FUNCTION_BLOCK fbChiniseMachine_v2_Laser IMPLEMENTS I_StationMachine
VAR_INPUT
	stSlaveParms				: stModTcpSlaveParams;
	bNextMachineWork			: BOOL;
	fbTCP_Send: REFERENCE TO FB_TCP_SendString;
	
END_VAR
VAR_OUTPUT
END_VAR
VAR
	I_PimSystem					: I_PIM;
	I_ModbusTcpCommunication 	: I_ModbusTcpCore;
	iWorkStep 					: INT;
	bServiceReset				: BOOL;
	stPimCommunicationData		: stPimMachineData;
	stModbusTcpData				: stModTcpQue;
	fbResetWaitTime				: TON;
	fbWorkEnded					: R_TRIG;					// Rising edgre reaction for end of cycle 
	iLastPartsRecord			: WORD;
	arReadArray					: ARRAY[0..GVL_ModbusTCP_Constants.iWriteRegisterLimit] OF INT;
	arWriteArray				: ARRAY[0..GVL_ModbusTCP_Constants.iWriteRegisterLimit] OF INT;
	rCommIntervalCounter		: REAL;
	nLastOperationStatus		: nModbusTCP_CommandStatus;
	fbCommunicationTimeout		: TON;
	bLastLifeBitState			: BOOL;
	stHMI						: stChiniseMachineHmiData;
	fbLifeBitPLC				: TON;
	stEthernetCommunication		: stInOutsEthernetCommunication;
	//Laser TCP
	fbLaserControl				:FB_LaserControl;
END_VAR

ACT_Background();
fbLaserControl(fbTCP_Send:=fbTCP_Send);

CASE iWorkStep OF
	0:	// Init
		iWorkStep := 5;
		
	5:	// Wait for next state
		I_PimSystem.mSetNewMachineState(nPIM_MachineStates._2_ReadyForNewOperation);	
		fbLaserControl.mRequestJobRefresh();
		iWorkStep := 10;
		
	10: // Start of work
		IF stPimCommunicationData.wGoodPartsAmount > iLastPartsRecord THEN
			IF I_PimSystem.mSetNewMachineState(nPIM_MachineStates._3_NewOperationStarted) THEN
				iLastPartsRecord := iLastPartsRecord +1;
				iWorkStep := 15;
				I_PimSystem.mSetNewMachineState(nPIM_MachineStates._4_OperationInProgress);
			END_IF
		END_IF
		IF fbLaserControl.stHMI_Laser.bEnableLaserTCPCOmmunication AND fbLaserControl.bJobRefreshError THEN
			mNewEvent(nEventClass:=nPIM_EventClasses.Error,nEvent:=nLaser_ErrorCodes.LaserTCPCommunicationError);
		END_IF
		
	15:	// Work ended
		iWorkStep := 5;
		I_PimSystem.mSetNewMachineState(nPIM_MachineStates._5_OperationEndedOK);
		
	90:	// Wysterowanie w przypadku błędu
		I_PimSystem.mSetNewMachineState(nPIM_MachineStates._8_WaitForReset);
		iWorkStep := 91;
		
	91:	// Oczekiwanie na reset
		IF I_PimSystem.mSetNewMachineState(nPIM_MachineStates._9_ResetInProgress) OR bServiceReset THEN
			bServiceReset := FALSE;
			stPimCommunicationData.bResetError := TRUE;
			fbCommunicationTimeout(IN:=FALSE);
			fbResetWaitTime(IN:=FALSE);
			iWorkStep := 92;
		END_IF
		
	92: // Wait some time
		fbResetWaitTime(IN:=TRUE,PT:=T#2S);
		IF fbResetWaitTime.Q THEN
			fbResetWaitTime(IN:=FALSE,PT:=T#2S);
			stPimCommunicationData.bResetError := FALSE;
			stPimCommunicationData.bConfirmError := TRUE;
			iWorkStep := 93;
		END_IF
		
	93:	// Check error state
		fbResetWaitTime(IN:=TRUE,PT:=T#2S);
		IF NOT stPimCommunicationData.bError THEN
			stPimCommunicationData.bConfirmError := FALSE;
			iWorkStep := 95;
			fbResetWaitTime(IN:=TRUE,PT:=T#2S);
		ELSIF fbResetWaitTime.Q THEN
			fbResetWaitTime(IN:=TRUE,PT:=T#2S);
			stPimCommunicationData.bResetError := FALSE;
			stPimCommunicationData.bConfirmError := FALSE;
			mNewEvent(nEventClass:=nPIM_EventClasses.Error,nEvent:=stPimCommunicationData.iErrorCode+stSlaveParms.iErrorOffset);
		END_IF
		
	95: // Potwierdzenie błędu itp
		I_PimSystem.mSetNewMachineState(nPIM_MachineStates._0_Standby_NotReady);
		stPimCommunicationData.bResetError := FALSE;
		stPimCommunicationData.bConfirmError := FALSE;
		iWorkStep := 5;
END_CASE

ACTION ACT_Background:
//Block parametrization form parameters
stModbusTcpData.sIpAdress 					:= stSlaveParms.sIpAdress;
stModbusTcpData.iPort 						:= stSlaveParms.iPort;
stModbusTcpData.iUnitId 					:= stSlaveParms.iUnitId;
stModbusTcpData.wRegistersReadQuantity		:= stSlaveParms.iRegisterReadAmount;
stModbusTcpData.wRegistersWriteQuantity		:= stSlaveParms.iRegisterWriteAmount;
stModbusTcpData.sMachineIndifiner			:= stSlaveParms.sMachineIdenfier;
stModbusTcpData.iRegisterReadStartAdress	:= stSlaveParms.iRegisterReadStartAdress;
stModbusTcpData.iRegisterWriteStartAdress	:= stSlaveParms.iRegisterWriteStartAdress;
//Rewrite signals from PIM System
//stMachineModbusParams.stPimData.bOfflineWorkAllow :=FALSE;
stPimCommunicationData.bStopPerform:=NOT bNextmachineWork OR (fbLaserControl.stHMI_Laser.bEnableLaserTCPCOmmunication AND NOT fbLaserControl.bJobRefreshed);
stPimCommunicationData.bTestMode:=I_PimSystem.prTestMode;
stPimCommunicationData.bWaitWithWork:=I_PimSystem.prPlcBlockWork;
stPimCommunicationData.bWorkAllow:=I_PimSystem.prWorkPermission ;
//Rewrite signals - signal for Lifebit
// Need to add iPartsCreatedInOneTime!!!

fbLifeBitPLC(IN:=NOT fbLifeBitPLC.Q ,PT:=T#500MS);

//Triggers
fbWorkEnded(CLK:=stPimCommunicationData.bCycleEnd);
//Data to send to slave

stEthernetCommunication.iProductID			:= stPimCommunicationData.iProductId;
stEthernetCommunication.iLifeBitPLC		:= BOOL_TO_INT(stPimCommunicationData.bLifeBitPLC);
stEthernetCommunication.iWorkAllow		:= BOOL_TO_INT(stPimCommunicationData.bWorkAllow);
stEthernetCommunication.iResetError		:= BOOL_TO_INT(stPimCommunicationData.bResetError);
stEthernetCommunication.iConfirmError		:= BOOL_TO_INT(stPimCommunicationData.bConfirmError);
stEthernetCommunication.iTestMode		:= BOOL_TO_INT(stPimCommunicationData.bTestMode);
stEthernetCommunication.iStopPerform		:= BOOL_TO_INT(stPimCommunicationData.bStopPerform);
stEthernetCommunication.iWaitWithWork		:= BOOL_TO_INT(stPimCommunicationData.bWaitWithWork);
stEthernetCommunication.iOfflineWorkAllow		:= BOOL_TO_INT(stPimCommunicationData.bOfflineWorkAllow);


//Data to read form slave
stPimCommunicationData.iActualWorkStep			:= stEthernetCommunication.iActualWorkStep;
stPimCommunicationData.wGoodPartsAmount			:= INT_TO_WORD(stEthernetCommunication.iGoodPartsAmountHighByte*256+stEthernetCommunication.iGoodPartsAmountLowByte);
stPimCommunicationData.wBadPartsAmount			:= INT_TO_WORD(stEthernetCommunication.iBadPartsAmountHighByte*256+stEthernetCommunication.iBadPartsAmountLowByte);
stPimCommunicationData.iCycleTime				:= stEthernetCommunication.iCycleTime;
stPimCommunicationData.iPartsCreatedInOneTime	:= stEthernetCommunication.iPartsCreatedInOneTime;
stPimCommunicationData.iErrorCode				:= stEthernetCommunication.iErrorCode;
stPimCommunicationData.bLifeBitMachine			:= INT_TO_BOOL(stEthernetCommunication.iLifeBitMachine);
stPimCommunicationData.bWorkInProgress			:= INT_TO_BOOL(stEthernetCommunication.iWorkInProgress);
stPimCommunicationData.bCycleEnd				:= INT_TO_BOOL(stEthernetCommunication.iCycleEnd);
stPimCommunicationData.bError					:= INT_TO_BOOL(stEthernetCommunication.iError);
stPimCommunicationData.bAlarm					:= INT_TO_BOOL(stEthernetCommunication.iAlarm);	
			
//Add command to que 
IF stSlaveParms.bCommunicationActive THEN
	rCommIntervalCounter := rCommIntervalCounter + 0.01;
ELSE
	rCommIntervalCounter := 0;
END_IF
IF rCommIntervalCounter >= stSlaveParms.rCommunicationCycleTime THEN
		rCommIntervalCounter := 0;
		//nLastOperationStatus := I_ModbusTcpCommunication.mAddToQue(stCommParams:=stModbusTcpData);
		stPimCommunicationData.bLifeBitPLC := NOT stPimCommunicationData.bLifeBitPLC;
END_IF

// Check of communication
IF stSlaveParms.bCommunicationActive THEN
	fbCommunicationTimeout(IN:=TRUE,PT:=T#10S);
	IF stPimCommunicationData.bLifeBitMachine <> bLastLifeBitState THEN
		bLastLifeBitState := stPimCommunicationData.bLifeBitMachine;
		fbCommunicationTimeout(IN:=FALSE);
	END_IF
	IF fbCommunicationTimeout.Q AND iWorkStep < 90 THEN
		mNewEvent(nEventClass:=nPIM_EventClasses.Error,nEvent:=nChiniseMachineErrorCodes.communicationError);
	END_IF
END_IF

// Check of Error
IF stPimCommunicationData.bError AND iWorkStep < 90 AND stSlaveParms.bCommunicationActive THEN
	mNewEvent(nEventClass:=nPIM_EventClasses.Error,nEvent:=stPimCommunicationData.iErrorCode+stSlaveParms.iErrorOffset);
	iWorkStep:=90;
END_IF

//Zabezpieczenie przed błędami w odczycie części do liczenia
IF (stPimCommunicationData.wGoodPartsAmount - iLastPartsRecord) > 5  OR (stPimCommunicationData.wGoodPartsAmount - iLastPartsRecord) < 0 THEN
	iLastPartsRecord := stPimCommunicationData.wGoodPartsAmount;
END_IF
//Parts reset
IF stPimCommunicationData.wGoodPartsAmount = 0  THEN
	iLastPartsRecord := 0;
END_IF


stHMI.nLastOperationStatus 		:= nLastOperationStatus;
stHMI.stModbusTcpData 			:= stModbusTcpData;
stHMI.stPimCommunicationData 	:= stPimCommunicationData;
END_ACTION

METHOD FB_init : BOOL
VAR_INPUT
	bInitRetains	: BOOL;
	bInCopyCode 	: BOOL;
	I_Pim			: I_PIM;
	I_ModbusCore	: I_ModbusTcpCore;
END_VAR
I_PimSystem := I_Pim;
I_ModbusTcpCommunication := I_ModbusCore;
stModbusTcpData.arRegisterReadArray := ADR(arReadArray);
stModbusTcpData.arRegisterWriteArray := ADR(arWriteArray);
END_METHOD

// Metoda TRUE kiedy dane wyjściowe są ok, jeśli nie FALSE (jeśli not bBusy i FALSE to błąd odczytu) 
METHOD mGetParamsData : BOOL
VAR_INPUT
	bTestParams:	BOOL;	// Jeśli TRUE metoda okresla czy ma dostęp do parametrów, jeśli tak zwraca TRUE, jeśli nie FALSE
END_VAR
VAR_OUTPUT
	bBusy:BOOL;		// Maszyna odświeża dane
	pMachineParametersStruct: POINTER TO BYTE;	// Wskaźnik do parametrów pracy maszyny
	uiMachineParametersSize: UINT;				// Rozmiar struktury parametrów pracy maszyny [bajty]
	wActualCRC16SumInMachine: WORD;				// Aktualna suma CRC16 obliczona z parametrów
END_VAR
IF bTestParams THEN
	mGetParamsData := FALSE;
ELSE
	pMachineParametersStruct := 0;
	uiMachineParametersSize := 0;
	bBusy := FALSE;
	mGetParamsData := TRUE;	
END_IF
END_METHOD

METHOD INTERNAL mNewEvent : BOOL
VAR_INPUT
	nEventClass:nPIM_EventClasses;
	nEvent: INT;
END_VAR
IF nEventClass = nPIM_EventClasses.AlarmAutoConfirm OR nEventClass = nPIM_EventClasses.Message THEN		// Alarm nieblokadowy
	I_PimSystem.mSetNewMachineState(nPIM_MachineStates._0_Initialization);
	iWorkStep := 90;
ELSE
	I_PimSystem.mSetNewMachineState(nPIM_MachineStates._7_ErrorOccurr);

	I_PimSystem.mNewEvent(iEventId := nEvent, nEventType := nEventClass, tMessageTime := T#0S);
	iWorkStep := 90;
END_IF
END_METHOD

END_FUNCTION_BLOCK

(* stored: Version 1.1.0.1, ProductVersion 3.1.4024.15
   POU fbChiniseMachine_v2_Laser: Id {4d39300c-1d2b-4451-b589-b239f8617dbc}, SpecialFunc None
   Action ACT_Background: Id {5427fb27-a0b5-485a-892f-7c195804c388}
   Method FB_init: Id {ee1b368b-e427-4ee6-8370-6c74fc8d581b}
   Method mGetParamsData: Id {27dd33e1-285e-44ef-ab65-5a1667fabeb0}
   Method mNewEvent: Id {e6d60a00-1681-4a7a-a5bf-b20ac586ef27} *)
